TYPE E_SabberLoggerLevel :
(
	Info,
	Warning,
	Error
);
END_TYPE

(* stored: Version 1.1.0.1, ProductVersion 3.1.0.36
   DUT E_SabberLoggerLevel: Id {90469d56-8c4e-4d5a-844e-f98202bff660} *)
